{attribute 'qualified_only'}
{attribute 'strict'}
TYPE E_CommState :
(
    eDisconnected := 0,
    eConnecting := 10,
    eConnected := 20,
    eDisconnecting := 30,
    eReconnectWait := 40
);
END_TYPE

(* stored: Version 1.1.0.1, ProductVersion 3.1.4026.18
   DUT E_CommState: Id {454aae8e-62f1-43e1-a34f-404d20f80024} *)
